// TwinCAT 3 PLC project ServerInterface
// ProgramVersion: 3.1.4023.0
// libraries:
//   Tc2_Standard, * (Beckhoff Automation GmbH)
//   Tc2_System, * (Beckhoff Automation GmbH)
//   Tc2_TcpIp, * (Beckhoff Automation GmbH)
//   Tc3_Module, * (Beckhoff Automation GmbH)
// project tree:
//   DUTs/ E_ServerPhases.TcDUT
//   / PlcTask.TcTTO
//   POUs/ MAIN.TcPOU
// real-time tasks:
//   TASK PlcTask: cycle T#10ms, priority 20, ADS port 350

CONFIGURATION ServerInterface
    RESOURCE PLC ON TwinCAT3
        TASK PlcTask(INTERVAL := T#10ms, PRIORITY := 20);
        PROGRAM MAIN WITH PlcTask : MAIN;
    END_RESOURCE
END_CONFIGURATION

// ---- DUTs/E_ServerPhases.TcDUT

TYPE E_ServerPhases :
(
	NO_PHASE := 0,
	INIT_PHASE := 10,
	START_PHASE := 20,
	RECEIVE_PHASE := 30
);
END_TYPE

// ---- POUs/MAIN.TcPOU
PROGRAM MAIN
VAR
	fbServerClientConnection : FB_ServerClientConnection;
	fbSocketSend : FB_SocketSend;
	fbSocketReceive : FB_SocketReceive;
	hServer : T_HSERVER; 
	
	bInit : BOOL := TRUE;
	
	ePhase : E_ServerPhases := INIT_PHASE;
	receiveBuffer : T_MAXSTRING;
END_VAR

F_CreateServerHnd(
	sSrvNetID := '127.0.0.1.1.1',
	sLocalHost := '',
	nLocalPort := 200,
	nMode :=  LISTEN_MODE_CLOSEALL,
	bEnable := bInit,
	hServer := hServer);

fbServerClientConnection(
	hServer := hServer,
	bEnable := NOT bInit,
	nRemotePort := 80,
	tReconnect := T#30MS);

fbSocketReceive(
	bExecute := (ePhase = RECEIVE_PHASE),
	tTimeout := T#30S,
	pDest := ADR(receiveBuffer),
	cbLen := SIZEOF(receiveBuffer),
	hSocket := fbServerClientConnection.hSocket);
	
	
CASE ePhase OF

	INIT_PHASE:
		bInit := FALSE;
		ePhase := START_PHASE;
		
	START_PHASE:
		IF fbServerClientConnection.eState = E_SocketConnectionState.eSOCKET_CONNECTED THEN
			ePhase := RECEIVE_PHASE;
		END_IF
		
	RECEIVE_PHASE:
		
		
END_CASE

END_PROGRAM
